FUNCTION_BLOCK TcoAxisRef EXTENDS Tc2_MC2.AXIS_REF

END_FUNCTION_BLOCK

(* stored: Version 1.1.0.1, ProductVersion 3.1.4024.12
   POU TcoAxisRef: Id {d42796a2-c667-02a2-28a2-386cb7a40c21}, SpecialFunc None *)
